ABB RobotStudio station: contour-following.rspag

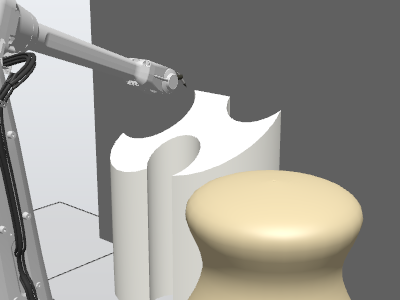
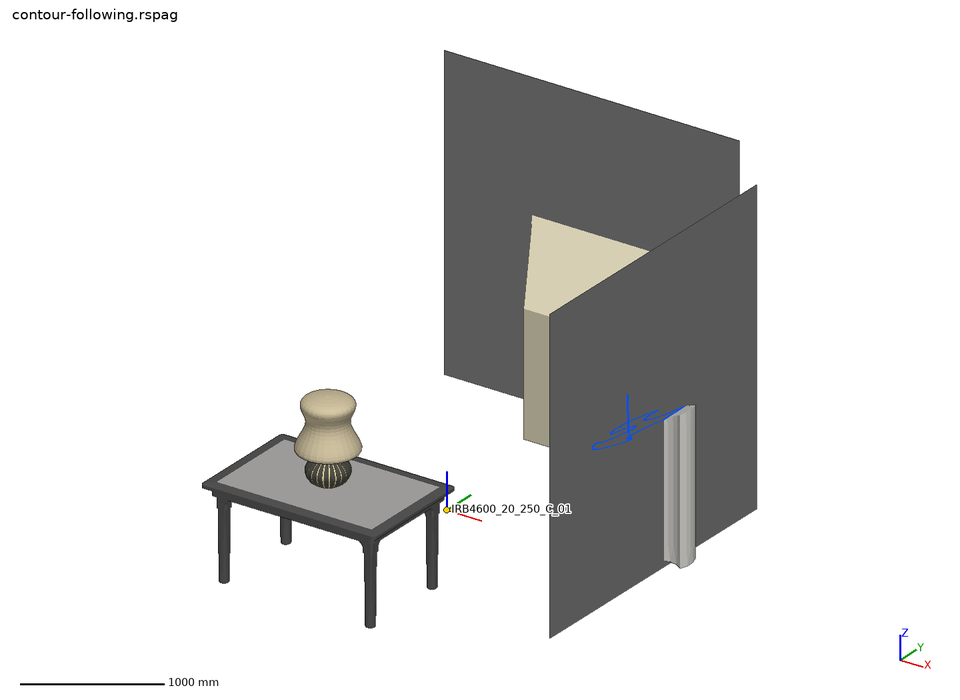
[picture v1: parts stored in the station drawn from their meshes, with robot base, taught points and paths (robot models come from the ABB library and are not in the file)]
--- station ---
Station PenPineappleApplePen (saved by RobotStudio 24.3.10885.0)
Controller Controller2
  mechanical unit ROB_1: IRB4600_20_250_C_01, 6 joints, base frame (0, 0, 0) mm
Layout (positions relative to the parent item):
  - IRB4600_20_250_C_01 [mechanism, from %ABB.RobotStudio.Models.IRB4600%\IRB4600_20_250_C_G_01.rslib] at (0, 0, 0) mm; joint values [0.1057, -0.1541, 0.5189, 0, -0.306, 0] (rad or m)
  - PenPineappleApplePen [mechanism, from Documents\PenPineappleApplePen.rslib] at (1296.51, 137.49, 1296.47) mm, rotated rx 180 ry 86.63 rz -173.95 deg
  - table2 [part] at (1845.28, -943.75, 534.88) mm, rotated rx 90 ry 0 rz 90 deg, size 984.1 x 770.9 x 1476.2 mm
  - trapez [part] at (500, 1748.7, 450) mm, rotated rx 90 ry 0 rz 90 deg, size 606.2 x 1387.4 x 1000 mm
  - krzywik [part] at (2000, 715.02, 706.25) mm, rotated rx 90 ry 0 rz 90 deg, size 823.5 x 1193.4 x 764.8 mm
  - lampa2 [part] at (112.5, -1435.82, 770.92) mm, rotated rx 90 ry 0 rz 90 deg, size 471.7 x 688.5 x 472.4 mm
  - Part_1 [part] at (1745, -1250, 0) mm, size 5 x 2500 x 2500 mm
  - Part_2 [part] at (-1250, 1750, 0) mm, size 2500 x 5 x 2500 mm
  - Frame_2 [frame] at (56.86, 0, 134.14) mm, rotated rx 0 ry 44.94 rz 0 deg
Attachment: PenPineappleApplePen is attached to IRB4600_20_250_C_01 / Link6
Attachment: trapez is attached to trapez
Attachment: krzywik is attached to krzywik
Attachment: lampa is attached to lampa2
Attachment: trapez is attached to Part_2
Attachment: lampa2 is attached to table2
Attachment: krzywik is attached to Part_1
Targets, tools, work objects and paths stored in the station and not in the controller backup, written as RAPID:
! task T_ROB1
MODULE CalibData
  TASK PERS wobjdata trapez:=[FALSE,TRUE,"",[[0,0,50],[1,0,0,0]],[[0,0,0],[1,0,0,0]]];
  TASK PERS wobjdata lampa:=[FALSE,TRUE,"",[[119.9,0,40.518],[1,0,0,0]],[[0,0,0],[1,0,0,0]]];
ENDMODULE

! task T_ROB1
MODULE Module1
  CONST robtarget Target_10:=[[-500,1748.705,1387.429],[0.270478686,-0.652549655,0.65678764,0.263913289],[1,2,1,0],[9E+09,9E+09,9E+09,9E+09,9E+09,9E+09]];
  CONST robtarget Target_20:=[[-150,1142.487,1006.377],[0.270478686,-0.652549655,0.65678764,0.263913289],[1,2,1,0],[9E+09,9E+09,9E+09,9E+09,9E+09,9E+09]];
  CONST robtarget Target_30:=[[150,1142.487,1006.377],[0.270478686,-0.652549655,0.65678764,0.263913289],[0,1,2,0],[9E+09,9E+09,9E+09,9E+09,9E+09,9E+09]];
  CONST robtarget Target_40:=[[500,1748.705,1387.429],[0.270478686,-0.652549655,0.65678764,0.263913289],[0,1,2,0],[9E+09,9E+09,9E+09,9E+09,9E+09,9E+09]];
  CONST robtarget above_trapez:=[[2.354624835,1375.15869908,1439.170310285],[0.270478686,-0.652549655,0.65678764,0.263913289],[1,2,1,0],[9E+09,9E+09,9E+09,9E+09,9E+09,9E+09]];
  CONST robtarget Target_300:=[[1764.521875862,134.170519561,1094.86146005],[0.355319487,-0.049345838,0.933252419,0.018787562],[0,-1,0,1],[9E+09,9E+09,9E+09,9E+09,9E+09,9E+09]];
  CONST robtarget Target_310:=[[1784.700794279,135.94993306,1106.51176403],[0.355319487,-0.049345838,0.933252419,0.018787562],[0,-1,0,1],[9E+09,9E+09,9E+09,9E+09,9E+09,9E+09]];
  CONST robtarget Target_320:=[[1804.953567722,135.525399506,1118.20470823],[0.355319487,-0.049345838,0.933252419,0.018787562],[0,-1,0,1],[9E+09,9E+09,9E+09,9E+09,9E+09,9E+09]];
  CONST robtarget Target_330:=[[1825.040194425,132.901949757,1129.801727564],[0.355319487,-0.049345838,0.933252419,0.018787562],[0,-1,0,1],[9E+09,9E+09,9E+09,9E+09,9E+09,9E+09]];
  CONST robtarget Target_340:=[[1844.722641512,128.110672521,1141.165393688],[0.355319487,-0.049345838,0.933252419,0.018787562],[0,-1,0,1],[9E+09,9E+09,9E+09,9E+09,9E+09,9E+09]];
  CONST robtarget Target_350:=[[1863.767665765,121.208345948,1152.161043566],[0.355319487,-0.049345838,0.933252419,0.018787562],[0,-1,0,1],[9E+09,9E+09,9E+09,9E+09,9E+09,9E+09]];
  CONST robtarget Target_360:=[[1881.949577625,112.276764789,1162.658375273],[0.355319487,-0.049345838,0.933252419,0.018787562],[0,-1,0,1],[9E+09,9E+09,9E+09,9E+09,9E+09,9E+09]];
  CONST robtarget Target_370:=[[1899.052915691,101.421771104,1172.53299211],[0.355319487,-0.049345838,0.933252419,0.018787562],[0,-1,0,1],[9E+09,9E+09,9E+09,9E+09,9E+09,9E+09]];
  CONST robtarget Target_380:=[[1914.875,88.772,1181.667876745],[0.355319487,-0.049345838,0.933252419,0.018787562],[0,-1,0,1],[9E+09,9E+09,9E+09,9E+09,9E+09,9E+09]];
  CONST robtarget Target_390:=[[1924.367037707,112.000280725,1187.14810727],[0.355319487,-0.049345838,0.933252419,0.018787562],[0,-1,0,1],[9E+09,9E+09,9E+09,9E+09,9E+09,9E+09]];
  CONST robtarget Target_400:=[[1930.986602832,136.204271363,1190.969914977],[0.355319487,-0.049345838,0.933252419,0.018787562],[0,-1,0,1],[9E+09,9E+09,9E+09,9E+09,9E+09,9E+09]];
  CONST robtarget Target_410:=[[1934.636942574,161.030201859,1193.07743961],[0.355319487,-0.049345838,0.933252419,0.018787562],[0,-1,0,1],[9E+09,9E+09,9E+09,9E+09,9E+09,9E+09]];
  CONST robtarget Target_420:=[[1935.264702885,186.11521177,1193.439877194],[0.355319487,-0.049345838,0.933252419,0.018787562],[0,-1,0,1],[9E+09,9E+09,9E+09,9E+09,9E+09,9E+09]];
  CONST robtarget Target_430:=[[1932.860708302,211.092653899,1192.051930274],[0.355319487,-0.049345838,0.933252419,0.018787562],[0,0,-1,1],[9E+09,9E+09,9E+09,9E+09,9E+09,9E+09]];
  CONST robtarget Target_440:=[[1927.460096059,235.597453279,1188.933885342],[0.355319487,-0.049345838,0.933252419,0.018787562],[0,0,-1,1],[9E+09,9E+09,9E+09,9E+09,9E+09,9E+09]];
  CONST robtarget Target_450:=[[1919.141802515,259.271443179,1184.131316326],[0.355319487,-0.049345838,0.933252419,0.018787562],[0,0,-1,1],[9E+09,9E+09,9E+09,9E+09,9E+09,9E+09]];
  CONST robtarget Target_460:=[[1908.027409406,281.768600134,1177.714418472],[0.355319487,-0.049345838,0.933252419,0.018787562],[0,0,-1,1],[9E+09,9E+09,9E+09,9E+09,9E+09,9E+09]];
  CONST robtarget Target_470:=[[1894.279366779,302.76010149,1169.77698236],[0.355319487,-0.049345838,0.933252419,0.018787562],[0,0,-1,1],[9E+09,9E+09,9E+09,9E+09,9E+09,9E+09]];
  CONST robtarget Target_480:=[[1878.098618597,321.939131536,1160.435023042],[0.355319487,-0.049345838,0.933252419,0.018787562],[0,0,-1,1],[9E+09,9E+09,9E+09,9E+09,9E+09,9E+09]];
  CONST robtarget Target_490:=[[1859.721665702,339.025365983,1149.825084341],[0.355319487,-0.049345838,0.933252419,0.018787562],[0,0,-1,1],[9E+09,9E+09,9E+09,9E+09,9E+09,9E+09]];
  CONST robtarget Target_500:=[[1839.417109075,353.76906923,1138.102243107],[0.355319487,-0.049345838,0.933252419,0.018787562],[0,0,-1,1],[9E+09,9E+09,9E+09,9E+09,9E+09,9E+09]];
  CONST robtarget Target_510:=[[1817.481723914,365.954744554,1125.43784258],[0.355319487,-0.049345838,0.933252419,0.018787562],[0,0,-1,1],[9E+09,9E+09,9E+09,9E+09,9E+09,9E+09]];
  CONST robtarget Target_520:=[[1794.236121912,375.404283845,1112.016988006],[0.355319487,-0.049345838,0.933252419,0.018787562],[0,0,-1,1],[9E+09,9E+09,9E+09,9E+09,9E+09,9E+09]];
  CONST robtarget Target_530:=[[1770.020065136,381.979570869,1098.035841107],[0.355319487,-0.049345838,0.933252419,0.018787562],[0,0,-1,1],[9E+09,9E+09,9E+09,9E+09,9E+09,9E+09]];
  CONST robtarget Target_1470:=[[-356.227701034,-1435.823,1008.367912023],[0,0.5726162,0,0.819823571],[-2,0,0,0],[9E+09,9E+09,9E+09,9E+09,9E+09,9E+09]];
  CONST robtarget Target_1480:=[[-356.632819707,-1435.823,1024.985425278],[0,0.7722597,0,0.635306978],[-2,0,0,0],[9E+09,9E+09,9E+09,9E+09,9E+09,9E+09]];
  CONST robtarget Target_1490:=[[-349.496807665,-1435.823,1046.554535488],[0,0.834440548,0,0.55109797],[-2,0,0,0],[9E+09,9E+09,9E+09,9E+09,9E+09,9E+09]];
  CONST robtarget Target_1500:=[[-337.487544389,-1435.823,1071.313546721],[0,0.856155357,0,0.516718497],[-2,0,0,0],[9E+09,9E+09,9E+09,9E+09,9E+09,9E+09]];
  CONST robtarget Target_1510:=[[-308.314339892,-1435.823,1124.876064439],[0,0.855906278,0,0.517130974],[-2,0,0,0],[9E+09,9E+09,9E+09,9E+09,9E+09,9E+09]];
  CONST robtarget Target_1520:=[[-285.046138139,-1435.823,1178.110750529],[0,0.805538472,0,0.592543476],[-2,0,0,0],[9E+09,9E+09,9E+09,9E+09,9E+09,9E+09]];
  CONST robtarget Target_1530:=[[-279.294170946,-1435.823,1203.768042628],[0,0.750595327,0,0.660762177],[-2,0,0,0],[9E+09,9E+09,9E+09,9E+09,9E+09,9E+09]];
  CONST robtarget Target_1540:=[[-278.820319707,-1435.823,1229.036477464],[0,0.672760595,0,0.739860245],[-2,0,0,0],[9E+09,9E+09,9E+09,9E+09,9E+09,9E+09]];
  CONST robtarget Target_1550:=[[-284.181369532,-1435.823,1254.504702787],[0,0.590226841,0,0.807237435],[-2,0,0,0],[9E+09,9E+09,9E+09,9E+09,9E+09,9E+09]];
  CONST robtarget Target_1560:=[[-316.030461305,-1435.823,1334.787935859],[0,0.640987484,0,0.767551331],[-2,0,0,0],[9E+09,9E+09,9E+09,9E+09,9E+09,9E+09]];
  CONST robtarget Target_1570:=[[-313.831298622,-1435.823,1361.259758709],[0,0.834769365,0,0.550599771],[-2,0,0,0],[9E+09,9E+09,9E+09,9E+09,9E+09,9E+09]];
  CONST robtarget Target_1580:=[[-305.449627822,-1435.823,1373.780481427],[0,0.918497838,0,0.395425999],[-2,0,0,0],[9E+09,9E+09,9E+09,9E+09,9E+09,9E+09]];
  CONST robtarget Target_1590:=[[-290.274693372,-1435.823,1385.522452993],[0,0.964723418,0,0.263265506],[-2,-1,0,0],[9E+09,9E+09,9E+09,9E+09,9E+09,9E+09]];
  CONST robtarget Target_1600:=[[-266.667771673,-1435.823,1396.219409162],[0,0.985506762,0,0.169636146],[-2,-1,0,0],[9E+09,9E+09,9E+09,9E+09,9E+09,9E+09]];
  CONST robtarget Target_1610:=[[-232.842282653,-1435.823,1405.5732495],[0,0.994311989,0,0.106506661],[-2,-1,1,0],[9E+09,9E+09,9E+09,9E+09,9E+09,9E+09]];
  CONST robtarget Target_1620:=[[-186.863789768,-1435.823,1413.254037383],[0,0.997988983,0,0.063387614],[-1,-1,1,0],[9E+09,9E+09,9E+09,9E+09,9E+09,9E+09]];
  CONST robtarget Target_1630:=[[-126.65,-1435.823,1418.9],[0,0.999455226,0,0.033003814],[-1,-1,1,0],[9E+09,9E+09,9E+09,9E+09,9E+09,9E+09]];
  CONST robtarget Target_1640:=[[-129.948583459,-1435.823,1468.791074825],[0,0.999455226,0,0.033003814],[-1,-1,1,0],[9E+09,9E+09,9E+09,9E+09,9E+09,9E+09]];
  CONST robtarget above_lamp:=[[-394.039408817,-1297.199647583,1588.358827541],[0.508942412,0.79207847,0.336817323,-0.011975388],[-2,-1,1,0],[9E+09,9E+09,9E+09,9E+09,9E+09,9E+09]];
  CONST robtarget back_trace:=[[-404.928368365,-1011.661568461,885.919207147],[0.385577292,0.834726208,0.074942636,0.385935112],[-2,0,0,0],[9E+09,9E+09,9E+09,9E+09,9E+09,9E+09]];
  CONST robtarget Target_1650:=[[1079.225,237.179079749,785.646448491],[0.101814374,0.888048773,0.379976418,0.237951952],[0,0,0,0],[9E+09,9E+09,9E+09,9E+09,9E+09,9E+09]];
  CONST robtarget Target_1660:=[[1104.225,237.179079749,742.345178302],[0.101814374,0.888048773,0.379976418,0.237951952],[0,-1,1,0],[9E+09,9E+09,9E+09,9E+09,9E+09,9E+09]];
  CONST robtarget Target_1670:=[[1135.277965809,264.790385883,760.273616471],[0.065302717,0.934674621,0.243713057,0.25044531],[0,-1,1,0],[9E+09,9E+09,9E+09,9E+09,9E+09,9E+09]];
  CONST robtarget Target_1680:=[[1173.212092282,281.751310408,782.174894602],[0.030064157,0.95938712,0.112200961,0.257067004],[0,-1,2,0],[9E+09,9E+09,9E+09,9E+09,9E+09,9E+09]];
  CONST robtarget Target_1690:=[[1214.495098447,286.482516812,806.009649324],[0.004378616,-0.965787589,0.016341217,-0.258782004],[0,0,2,0],[9E+09,9E+09,9E+09,9E+09,9E+09,9E+09]];
  CONST robtarget Target_1700:=[[1255.282868444,278.543453224,829.558479312],[0.038945016,-0.954928058,0.14534478,-0.255872202],[0,0,2,0],[9E+09,9E+09,9E+09,9E+09,9E+09,9E+09]];
  CONST robtarget Target_1710:=[[1291.777400916,258.673374924,850.628607458],[0.074493857,-0.925051588,0.278014857,-0.247866826],[0,0,2,0],[9E+09,9E+09,9E+09,9E+09,9E+09,9E+09]];
  CONST robtarget Target_1720:=[[1320.580464386,228.722507712,867.258063906],[0.111291008,-0.872067838,0.415343698,-0.233669873],[0,0,2,0],[9E+09,9E+09,9E+09,9E+09,9E+09,9E+09]];
  CONST robtarget Target_1730:=[[1339.010027592,191.479761948,877.898377184],[0.148334096,-0.79154936,0.553590384,-0.212095012],[0,0,2,0],[9E+09,9E+09,9E+09,9E+09,9E+09,9E+09]];
  CONST robtarget Target_1740:=[[1345.35,150.413039874,881.558761961],[0.183012702,-0.683012702,0.683012702,-0.183012702],[0,0,2,0],[9E+09,9E+09,9E+09,9E+09,9E+09,9E+09]];
  CONST robtarget Target_1750:=[[1339.010027592,109.346317801,877.898377184],[0.212095012,-0.553590384,0.79154936,-0.148334096],[0,0,2,0],[9E+09,9E+09,9E+09,9E+09,9E+09,9E+09]];
  CONST robtarget Target_1760:=[[1320.580464386,72.103572037,867.258063906],[0.233669873,-0.415343698,0.872067838,-0.111291008],[-1,1,2,0],[9E+09,9E+09,9E+09,9E+09,9E+09,9E+09]];
  CONST robtarget Target_1770:=[[1291.777400916,42.152704825,850.628607458],[0.247866826,-0.278014857,0.925051588,-0.074493857],[-1,1,2,0],[9E+09,9E+09,9E+09,9E+09,9E+09,9E+09]];
  CONST robtarget Target_1780:=[[1255.282868444,22.282626525,829.558479312],[0.255872202,-0.14534478,0.954928058,-0.038945016],[-1,1,2,0],[9E+09,9E+09,9E+09,9E+09,9E+09,9E+09]];
  CONST robtarget Target_1790:=[[1214.495098447,14.343562937,806.009649324],[0.258782004,-0.016341217,0.965787589,-0.004378616],[0,1,2,0],[9E+09,9E+09,9E+09,9E+09,9E+09,9E+09]];
  CONST robtarget Target_1800:=[[1173.212092282,19.074769341,782.174894602],[0.257067004,0.112200961,0.95938712,0.030064157],[0,2,1,0],[9E+09,9E+09,9E+09,9E+09,9E+09,9E+09]];
  CONST robtarget Target_1810:=[[1135.277965809,36.035693866,760.273616471],[0.25044531,0.243713057,0.934674621,0.065302717],[0,2,1,0],[9E+09,9E+09,9E+09,9E+09,9E+09,9E+09]];
  CONST robtarget Target_1820:=[[1104.225,63.647,742.345178302],[0.237951952,0.379976418,0.888048773,0.101814374],[0,2,1,0],[9E+09,9E+09,9E+09,9E+09,9E+09,9E+09]];
  CONST robtarget Target_1830:=[[1115.168705531,24.942095166,748.663529636],[0.145865677,-0.797913008,0.544378117,-0.213800146],[-1,0,2,0],[9E+09,9E+09,9E+09,9E+09,9E+09,9E+09]];
  CONST robtarget Target_1840:=[[1130.03531583,-12.431936557,757.246771094],[0.133473684,-0.827573947,0.498130569,-0.221747771],[-1,0,2,0],[9E+09,9E+09,9E+09,9E+09,9E+09,9E+09]];
  CONST robtarget Target_1850:=[[1148.667140429,-48.078667979,768.003860042],[0.120964856,-0.853936951,0.45144699,-0.228811716],[-1,0,2,0],[9E+09,9E+09,9E+09,9E+09,9E+09,9E+09]];
  CONST robtarget Target_1860:=[[1170.86655115,-81.619993425,780.820695798],[0.108438136,-0.877059483,0.404696634,-0.23500738],[-1,0,2,0],[9E+09,9E+09,9E+09,9E+09,9E+09,9E+09]];
  CONST robtarget Target_1870:=[[1196.398078347,-112.700139306,795.561329898],[0.095969627,-0.897068332,0.358163523,-0.240368735],[-1,0,2,0],[9E+09,9E+09,9E+09,9E+09,9E+09,9E+09]];
  CONST robtarget Target_1880:=[[1224.990908541,-140.989437821,812.069408107],[0.083611988,-0.914134086,0.312044187,-0.24494149],[-1,0,2,0],[9E+09,9E+09,9E+09,9E+09,9E+09,9E+09]];
  CONST robtarget Target_1890:=[[1256.341756944,-166.187823749,830.169828872],[0.071395991,-0.928447766,0.266453464,-0.248776829],[-1,0,2,0],[9E+09,9E+09,9E+09,9E+09,9E+09,9E+09]];
  CONST robtarget Target_1900:=[[1290.118084407,-188.028017249,849.670600625],[0.059333361,-0.940201676,0.221435117,-0.25192628],[-1,0,2,0],[9E+09,9E+09,9E+09,9E+09,9E+09,9E+09]];
  CONST robtarget Target_1910:=[[1325.96162467,-206.2783589,870.364878245],[0.047420169,-0.949575029,0.17697448,-0.254437862],[-1,0,2,0],[9E+09,9E+09,9E+09,9E+09,9E+09,9E+09]];
  CONST robtarget Target_1920:=[[1363.492184502,-220.745266921,892.033157066],[0.035640235,-0.956723957,0.133011169,-0.256353412],[-1,0,1,0],[9E+09,9E+09,9E+09,9E+09,9E+09,9E+09]];
  CONST robtarget Target_1930:=[[1402.311676416,-231.275290496,914.445601173],[0.023968254,-0.96177506,0.089450741,-0.257706851],[-1,0,1,0],[9E+09,9E+09,9E+09,9E+09,9E+09,9E+09]];
  CONST robtarget Target_1940:=[[1442.008341196,-237.756737429,937.36448127],[0.012372518,-0.964821529,0.046174865,-0.25852315],[-1,0,1,0],[9E+09,9E+09,9E+09,9E+09,9E+09,9E+09]];
  CONST robtarget Target_1950:=[[1482.161115432,-240.120858867,960.546696283],[0.000817262,-0.965921011,0.003050063,-0.258817755],[-1,-1,1,0],[9E+09,9E+09,9E+09,9E+09,9E+09,9E+09]];
  CONST robtarget Target_1960:=[[1522.34409775,-238.342578523,983.746351942],[0.010735293,0.965094568,0.04006466,0.25859631],[-1,-1,1,0],[9E+09,9E+09,9E+09,9E+09,9E+09,9E+09]];
  CONST robtarget Target_1970:=[[1562.131066361,-232.440758656,1006.717368979],[0.022323059,0.962326355,0.08331079,0.25785457],[-1,-1,1,0],[9E+09,9E+09,9E+09,9E+09,9E+09,9E+09]];
  CONST robtarget Target_1980:=[[1601.1,-222.478,1029.216093306],[0.033982204,0.957563862,0.126823313,0.256578463],[-1,-1,1,0],[9E+09,9E+09,9E+09,9E+09,9E+09,9E+09]];
  CONST robtarget Target_1990:=[[1565.485723439,-203.289964368,1008.654181146],[0.249518515,0.256612319,0.931215775,0.068759064],[-1,-2,1,0],[9E+09,9E+09,9E+09,9E+09,9E+09,9E+09]];
  CONST robtarget Target_2000:=[[1534.859704885,-176.858838892,990.97224109],[0.240877448,0.353371284,0.898966872,0.09468555],[-1,-2,1,0],[9E+09,9E+09,9E+09,9E+09,9E+09,9E+09]];
  CONST robtarget Target_2010:=[[1510.669355527,-144.433780614,977.005936376],[0.228741176,0.45194461,0.853673691,0.121098193],[-1,-1,1,0],[9E+09,9E+09,9E+09,9E+09,9E+09,9E+09]];
  CONST robtarget Target_2020:=[[1494.057931457,-107.547224842,967.415326218],[0.212747139,0.550094071,0.793983133,0.147397262],[-1,-1,1,0],[9E+09,9E+09,9E+09,9E+09,9E+09,9E+09]];
  CONST robtarget Target_2030:=[[1485.810502435,-67.942460975,962.653670852],[0.192899661,0.644003393,0.719911336,0.172560189],[0,-1,1,0],[9E+09,9E+09,9E+09,9E+09,9E+09,9E+09]];
  CONST robtarget Target_2040:=[[1486.31684884,-27.491243198,962.946010085],[0.169765377,0.729107632,0.633573014,0.195363801],[0,-1,1,0],[9E+09,9E+09,9E+09,9E+09,9E+09,9E+09]];
  CONST robtarget Target_2050:=[[1495.553040316,11.89467019,968.27852772],[0.144410213,0.80159194,0.538946253,0.214785913],[0,-1,1,0],[9E+09,9E+09,9E+09,9E+09,9E+09,9E+09]];
  CONST robtarget Target_2060:=[[1513.082566748,48.353868061,978.399204525],[0.118053068,0.859594046,0.440580048,0.23032753],[0,-1,1,0],[9E+09,9E+09,9E+09,9E+09,9E+09,9E+09]];
  CONST robtarget Target_2070:=[[1538.076968094,80.163258307,992.82972887],[0.091674424,0.903303545,0.342133609,0.242039456],[0,-1,1,0],[9E+09,9E+09,9E+09,9E+09,9E+09,9E+09]];
  CONST robtarget Target_2080:=[[1569.354988092,105.819502603,1010.888102135],[0.065822324,0.934166832,0.245652257,0.250309248],[0,-1,1,0],[9E+09,9E+09,9E+09,9E+09,9E+09,9E+09]];
  CONST robtarget Target_2090:=[[1605.43840142,124.110065441,1031.720870534],[0.040637159,0.953945472,0.151659942,0.255608919],[0,-1,1,0],[9E+09,9E+09,9E+09,9E+09,9E+09,9E+09]];
  CONST robtarget Target_2100:=[[1644.621875862,134.170519561,1054.34346005],[0.015977034,0.964083664,0.059627104,0.258325439],[0,-1,1,0],[9E+09,9E+09,9E+09,9E+09,9E+09,9E+09]];
  CONST robtarget Target_2110:=[[1685.053567722,135.525399506,1077.68670823],[0.008454424,-0.965410354,0.031552341,-0.258680925],[0,0,2,0],[9E+09,9E+09,9E+09,9E+09,9E+09,9E+09]];
  CONST robtarget Target_2120:=[[1724.822641512,128.110672521,1100.647393688],[0.033008401,-0.958038186,0.123189029,-0.256705558],[0,0,2,0],[9E+09,9E+09,9E+09,9E+09,9E+09,9E+09]];
  CONST robtarget Target_2130:=[[1762.049577625,112.276764789,1122.140375273],[0.058007536,-0.941353307,0.216487073,-0.252234858],[0,0,2,0],[9E+09,9E+09,9E+09,9E+09,9E+09,9E+09]];
  CONST robtarget Target_2140:=[[1794.975,88.772,1141.149876745],[0.083653614,-0.914081041,0.312199539,-0.244927277],[0,0,2,0],[9E+09,9E+09,9E+09,9E+09,9E+09,9E+09]];
  CONST robtarget Target_2150:=[[1811.086602832,136.204271363,1150.451914977],[0.160061595,0.759062655,0.597358006,0.203390226],[0,-1,1,0],[9E+09,9E+09,9E+09,9E+09,9E+09,9E+09]];
  CONST robtarget Target_2160:=[[1815.364702885,186.11521177,1152.921877194],[0.186720933,0.668887119,0.69685201,0.179227763],[0,-1,1,0],[9E+09,9E+09,9E+09,9E+09,9E+09,9E+09]];
  CONST robtarget Target_2170:=[[1807.560096059,235.597453279,1148.415885342],[0.209655409,0.566385989,0.782444639,0.151762668],[0,-1,1,0],[9E+09,9E+09,9E+09,9E+09,9E+09,9E+09]];
  CONST robtarget Target_2180:=[[1788.127409406,281.768600134,1137.196418472],[0.227916914,0.457707976,0.850597502,0.122642482],[0,-1,1,0],[9E+09,9E+09,9E+09,9E+09,9E+09,9E+09]];
  CONST robtarget Target_2190:=[[1758.198618597,321.939131536,1119.917023042],[0.241413165,0.348242177,0.900966197,0.09331121],[0,-1,1,0],[9E+09,9E+09,9E+09,9E+09,9E+09,9E+09]];
  CONST robtarget Target_2200:=[[1719.517109075,353.76906923,1097.584243107],[0.250629262,0.241064801,0.935361141,0.064593119],[0,-2,1,0],[9E+09,9E+09,9E+09,9E+09,9E+09,9E+09]];
  CONST robtarget Target_2210:=[[1674.336121912,375.404283845,1071.498988006],[0.25620536,0.136926686,0.95617142,0.036689395],[0,-2,1,0],[9E+09,9E+09,9E+09,9E+09,9E+09,9E+09]];
  CONST robtarget Target_2220:=[[1625.2875,385.5845,1043.180752942],[0.258648972,0.035011232,0.965291104,0.009381231],[0,-2,1,0],[9E+09,9E+09,9E+09,9E+09,9E+09,9E+09]];
  CONST robtarget Target_2230:=[[1601.044864766,356.220958453,1029.184260964],[0.242378357,-0.338775461,0.904568344,-0.090774611],[0,-3,2,0],[9E+09,9E+09,9E+09,9E+09,9E+09,9E+09]];
  CONST robtarget Target_2240:=[[1571.827205325,331.802700693,1012.31543742],[0.249492039,-0.256970612,0.931116967,-0.068855068],[0,-3,2,0],[9E+09,9E+09,9E+09,9E+09,9E+09,9E+09]];
  CONST robtarget Target_2250:=[[1538.626094744,313.158420299,993.146767289],[0.25443798,-0.176972116,0.949575469,-0.047419536],[0,-3,2,0],[9E+09,9E+09,9E+09,9E+09,9E+09,9E+09]];
  CONST robtarget Target_2260:=[[1502.568294293,300.920856738,972.328786492],[0.257468504,-0.098547878,0.960885538,-0.026405824],[0,-2,1,0],[9E+09,9E+09,9E+09,9E+09,9E+09,9E+09]];
  CONST robtarget Target_2270:=[[1464.877514033,295.505321802,950.568004363],[0.258757227,-0.021110286,0.965695116,-0.005656484],[0,-2,1,0],[9E+09,9E+09,9E+09,9E+09,9E+09,9E+09]];
  CONST robtarget Target_2280:=[[1426.832883206,297.095604975,928.602926514],[0.25838206,0.056106136,0.964294977,0.015033594],[0,-2,1,0],[9E+09,9E+09,9E+09,9E+09,9E+09,9E+09]];
  CONST robtarget Target_2290:=[[1389.725539846,305.63773609,907.178991836],[0.256320082,0.133902818,0.95659957,0.035879152],[0,-2,1,0],[9E+09,9E+09,9E+09,9E+09,9E+09,9E+09]];
  CONST robtarget Target_2300:=[[1354.814812829,320.841816939,887.023274195],[0.25244889,0.212983924,0.942152084,0.057068871],[0,-2,1,0],[9E+09,9E+09,9E+09,9E+09,9E+09,9E+09]];
  CONST robtarget Target_2310:=[[1323.285483462,342.191859676,868.819807398],[0.246556037,0.293800792,0.920159658,0.078723685],[0,-2,1,0],[9E+09,9E+09,9E+09,9E+09,9E+09,9E+09]];
  CONST robtarget Target_2320:=[[1296.20757701,368.96329814,853.186370819],[0.238364885,0.376354326,0.889589862,0.100843838],[0,-2,1,0],[9E+09,9E+09,9E+09,9E+09,9E+09,9E+09]];
  CONST robtarget Target_2330:=[[1274.500048766,400.247577783,840.653523543],[0.227589702,0.459970159,0.849376333,0.123248633],[0,-1,1,0],[9E+09,9E+09,9E+09,9E+09,9E+09,9E+09]];
  CONST robtarget Target_2340:=[[1258.899597041,434.982989703,831.646598541],[0.214028605,0.543126297,0.798765627,0.145530253],[0,-1,1,0],[9E+09,9E+09,9E+09,9E+09,9E+09,9E+09]];
  CONST robtarget Target_2350:=[[1249.935661499,471.990702344,826.471267943],[0.197680828,0.623482494,0.737754893,0.167061631],[0,-1,1,0],[9E+09,9E+09,9E+09,9E+09,9E+09,9E+09]];
  CONST robtarget Target_2360:=[[1247.912455319,510.014768039,825.30316931],[0.178837583,0.698246829,0.667430946,0.187094674],[0,-1,1,0],[9E+09,9E+09,9E+09,9E+09,9E+09,9E+09]];
  CONST robtarget Target_2370:=[[1252.898640973,547.764746686,828.181944939],[0.158077387,0.764832237,0.589952838,0.20493618],[0,-1,1,0],[9E+09,9E+09,9E+09,9E+09,9E+09,9E+09]];
  CONST robtarget Target_2380:=[[1264.725,583.9595,835.009896507],[0.136140408,0.821501337,0.508082921,0.22012062],[0,-1,1,0],[9E+09,9E+09,9E+09,9E+09,9E+09,9E+09]];
  CONST robtarget Target_2390:=[[1234.428871964,582.733933377,817.51841883],[0.258505543,-0.047528015,0.964755819,-0.012735093],[0,-2,1,0],[9E+09,9E+09,9E+09,9E+09,9E+09,9E+09]];
  CONST robtarget Target_2400:=[[1204.634785103,577.106342805,800.316794761],[0.257164531,-0.109043723,0.959751097,-0.029218177],[0,-2,1,0],[9E+09,9E+09,9E+09,9E+09,9E+09,9E+09]];
  CONST robtarget Target_2410:=[[1175.978894374,567.196887017,783.772308534],[0.254719351,-0.171241772,0.950625561,-0.045884095],[0,-2,1,0],[9E+09,9E+09,9E+09,9E+09,9E+09,9E+09]];
  CONST robtarget Target_2420:=[[1149.073052289,553.217149921,768.238213364],[0.251081735,-0.234414993,0.937049792,-0.062811308],[0,-2,1,0],[9E+09,9E+09,9E+09,9E+09,9E+09,9E+09]];
  CONST robtarget Target_2430:=[[1124.491744818,535.46562293,754.046188878],[0.24613106,-0.298722627,0.918573619,-0.080042487],[0,-3,1,0],[9E+09,9E+09,9E+09,9E+09,9E+09,9E+09]];
  CONST robtarget Target_2440:=[[1102.759825117,514.321331652,741.499259189],[0.239725003,-0.364123117,0.894665892,-0.097566495],[0,-3,1,0],[9E+09,9E+09,9E+09,9E+09,9E+09,9E+09]];
  CONST robtarget Target_2450:=[[1084.34130702,490.235743044,730.865322808],[0.231718435,-0.430301818,0.864784972,-0.115299025],[0,-3,2,0],[9E+09,9E+09,9E+09,9E+09,9E+09,9E+09]];
  CONST robtarget Target_2460:=[[1069.629457541,463.723125813,722.371432551],[0.221992238,-0.496611654,0.828486311,-0.133066692],[0,-3,2,0],[9E+09,9E+09,9E+09,9E+09,9E+09,9E+09]];
  CONST robtarget Target_2470:=[[1058.93839995,435.349569901,716.198947572],[0.210490143,-0.562057232,0.785559909,-0.150602781],[0,-3,2,0],[9E+09,9E+09,9E+09,9E+09,9E+09,9E+09]];
  CONST robtarget Target_2480:=[[1052.496406698,405.720899487,712.479661035],[0.19725541,-0.625356329,0.736167212,-0.167563723],[0,-4,2,0],[9E+09,9E+09,9E+09,9E+09,9E+09,9E+09]];
  CONST robtarget Target_2490:=[[1050.441025414,375.469737604,711.292986097],[0.182453249,-0.685094245,0.680924795,-0.18357045],[0,-4,2,0],[9E+09,9E+09,9E+09,9E+09,9E+09,9E+09]];
  CONST robtarget Target_2500:=[[1052.816142018,345.241998545,712.664260308],[0.166364969,-0.739944323,0.620882518,-0.198267484],[0,-4,2,0],[9E+09,9E+09,9E+09,9E+09,9E+09,9E+09]];
  CONST robtarget Target_2510:=[[1059.571043691,315.683096486,716.564204607],[0.149349844,-0.788884587,0.557381207,-0.211380988],[0,-4,2,0],[9E+09,9E+09,9E+09,9E+09,9E+09,9E+09]];
  CONST robtarget Target_2520:=[[1070.561501673,287.424164785,722.909548481],[0.131786232,-0.831332116,0.491832913,-0.222754769],[0,-4,2,0],[9E+09,9E+09,9E+09,9E+09,9E+09,9E+09]];
  CONST robtarget Target_2530:=[[1085.552850798,261.068580198,731.564807934],[0.114013243,-0.867156107,0.425503217,-0.232353779],[0,-4,2,0],[9E+09,9E+09,9E+09,9E+09,9E+09,9E+09]];
  CONST robtarget Target_2540:=[[1104.225,237.179079749,742.345178302],[0.096291106,-0.896588379,0.3593633,-0.240240132],[0,-4,2,0],[9E+09,9E+09,9E+09,9E+09,9E+09,9E+09]];
  CONST robtarget Target_2550:=[[1079.225,237.179079749,785.646448491],[0.096291106,-0.896588379,0.3593633,-0.240240132],[0,-4,2,0],[9E+09,9E+09,9E+09,9E+09,9E+09,9E+09]];
  LOCAL PROC Path_10()
    MoveL above_trapez,v1000,fine,PenPineappleApplePen\WObj:=trapez;
    MoveL Target_10,v1000,fine,PenPineappleApplePen\WObj:=trapez;
    MoveL Target_20,v300,fine,PenPineappleApplePen\WObj:=trapez;
    MoveL Target_30,v300,fine,PenPineappleApplePen\WObj:=trapez;
    MoveL Target_40,v300,fine,PenPineappleApplePen\WObj:=trapez;
    MoveL Target_10,v300,fine,PenPineappleApplePen\WObj:=trapez;
    MoveL above_trapez,v1000,fine,PenPineappleApplePen\WObj:=trapez;
  ENDPROC
  PROC Path_20()
    MoveL above_krzywik,v1000,z100,PenPineappleApplePen\WObj:=krzywik;
    MoveL Target_50,v1000,z100,PenPineappleApplePen\WObj:=krzywik;
    MoveL Target_60,v300,fine,PenPineappleApplePen\WObj:=krzywik;
    MoveL Target_70,v300,z100,PenPineappleApplePen\WObj:=krzywik;
    MoveL Target_80,v300,z100,PenPineappleApplePen\WObj:=krzywik;
    MoveL Target_90,v300,z100,PenPineappleApplePen\WObj:=krzywik;
    MoveL Target_100,v300,z100,PenPineappleApplePen\WObj:=krzywik;
    MoveL Target_110,v300,z100,PenPineappleApplePen\WObj:=krzywik;
    MoveL Target_120,v300,z100,PenPineappleApplePen\WObj:=krzywik;
    MoveL Target_130,v300,z100,PenPineappleApplePen\WObj:=krzywik;
    MoveL Target_140,v300,z100,PenPineappleApplePen\WObj:=krzywik;
    MoveL Target_150,v300,z100,PenPineappleApplePen\WObj:=krzywik;
    MoveL Target_160,v300,z100,PenPineappleApplePen\WObj:=krzywik;
    MoveL Target_170,v300,z100,PenPineappleApplePen\WObj:=krzywik;
    MoveL Target_180,v300,z100,PenPineappleApplePen\WObj:=krzywik;
    MoveL Target_190,v300,z100,PenPineappleApplePen\WObj:=krzywik;
    MoveL Target_200,v300,z100,PenPineappleApplePen\WObj:=krzywik;
    MoveL Target_210,v300,z100,PenPineappleApplePen\WObj:=krzywik;
    MoveL Target_220,v300,z100,PenPineappleApplePen\WObj:=krzywik;
    MoveL Target_230,v300,z100,PenPineappleApplePen\WObj:=krzywik;
    MoveL Target_240,v300,z100,PenPineappleApplePen\WObj:=krzywik;
    MoveL Target_250,v300,z100,PenPineappleApplePen\WObj:=krzywik;
    MoveL Target_260,v300,z100,PenPineappleApplePen\WObj:=krzywik;
    MoveL Target_270,v300,z100,PenPineappleApplePen\WObj:=krzywik;
    MoveL Target_280,v300,z100,PenPineappleApplePen\WObj:=krzywik;
    MoveL Target_290,v300,z100,PenPineappleApplePen\WObj:=krzywik;
    MoveL Target_540,v300,z100,PenPineappleApplePen\WObj:=krzywik;
    MoveL Target_550,v300,z100,PenPineappleApplePen\WObj:=krzywik;
    MoveL Target_560,v300,z100,PenPineappleApplePen\WObj:=krzywik;
    MoveL Target_570,v300,z100,PenPineappleApplePen\WObj:=krzywik;
    MoveL Target_580,v300,z100,PenPineappleApplePen\WObj:=krzywik;
    MoveL Target_590,v300,z100,PenPineappleApplePen\WObj:=krzywik;
    MoveL Target_600,v300,z100,PenPineappleApplePen\WObj:=krzywik;
    MoveL Target_610,v300,z100,PenPineappleApplePen\WObj:=krzywik;
    MoveL Target_620,v300,z100,PenPineappleApplePen\WObj:=krzywik;
    MoveL Target_630,v300,z100,PenPineappleApplePen\WObj:=krzywik;
    MoveL Target_640,v300,z100,PenPineappleApplePen\WObj:=krzywik;
    MoveL Target_650,v300,z100,PenPineappleApplePen\WObj:=krzywik;
    MoveL Target_660,v300,z100,PenPineappleApplePen\WObj:=krzywik;
    MoveL Target_670,v300,z100,PenPineappleApplePen\WObj:=krzywik;
    MoveL Target_680,v300,z100,PenPineappleApplePen\WObj:=krzywik;
    MoveL Target_690,v300,z100,PenPineappleApplePen\WObj:=krzywik;
    MoveL Target_700,v300,z100,PenPineappleApplePen\WObj:=krzywik;
    MoveL Target_710,v300,z100,PenPineappleApplePen\WObj:=krzywik;
    MoveL Target_720,v300,z100,PenPineappleApplePen\WObj:=krzywik;
    MoveL Target_730,v300,z100,PenPineappleApplePen\WObj:=krzywik;
    MoveL Target_740,v300,z100,PenPineappleApplePen\WObj:=krzywik;
    MoveL Target_750,v300,z100,PenPineappleApplePen\WObj:=krzywik;
    MoveL Target_760,v300,z100,PenPineappleApplePen\WObj:=krzywik;
    MoveL Target_770,v300,z100,PenPineappleApplePen\WObj:=krzywik;
    MoveL Target_780,v300,z100,PenPineappleApplePen\WObj:=krzywik;
    MoveL Target_790,v300,z100,PenPineappleApplePen\WObj:=krzywik;
    MoveL Target_800,v300,z100,PenPineappleApplePen\WObj:=krzywik;
    MoveL Target_810,v300,z100,PenPineappleApplePen\WObj:=krzywik;
    MoveL Target_820,v300,z100,PenPineappleApplePen\WObj:=krzywik;
    MoveL Target_830,v300,z100,PenPineappleApplePen\WObj:=krzywik;
    MoveL Target_840,v300,z100,PenPineappleApplePen\WObj:=krzywik;
    MoveL Target_850,v300,z100,PenPineappleApplePen\WObj:=krzywik;
    MoveL Target_860,v300,z100,PenPineappleApplePen\WObj:=krzywik;
    MoveL Target_870,v300,z100,PenPineappleApplePen\WObj:=krzywik;
    MoveL Target_880,v300,z100,PenPineappleApplePen\WObj:=krzywik;
    MoveL Target_890,v300,z100,PenPineappleApplePen\WObj:=krzywik;
    MoveL Target_900,v300,z100,PenPineappleApplePen\WObj:=krzywik;
    MoveL Target_910,v300,z100,PenPineappleApplePen\WObj:=krzywik;
    MoveL Target_920,v300,z100,PenPineappleApplePen\WObj:=krzywik;
    MoveL Target_930,v300,z100,PenPineappleApplePen\WObj:=krzywik;
    MoveL Target_940,v300,z100,PenPineappleApplePen\WObj:=krzywik;
    MoveL Target_950,v300,z100,PenPineappleApplePen\WObj:=krzywik;
    MoveL Target_960,v300,z100,PenPineappleApplePen\WObj:=krzywik;
    MoveL Target_970,v300,z100,PenPineappleApplePen\WObj:=krzywik;
    MoveL Target_980,v300,z100,PenPineappleApplePen\WObj:=krzywik;
    MoveL Target_990,v300,z100,PenPineappleApplePen\WObj:=krzywik;
    MoveL Target_1000,v300,z100,PenPineappleApplePen\WObj:=krzywik;
    MoveL Target_1010,v300,z100,PenPineappleApplePen\WObj:=krzywik;
    MoveL Target_1020,v300,z100,PenPineappleApplePen\WObj:=krzywik;
    MoveL Target_1030,v300,z100,PenPineappleApplePen\WObj:=krzywik;
    MoveL Target_1040,v300,z100,PenPineappleApplePen\WObj:=krzywik;
    MoveL Target_1050,v300,z100,PenPineappleApplePen\WObj:=krzywik;
    MoveL Target_1060,v300,z100,PenPineappleApplePen\WObj:=krzywik;
    MoveL Target_1070,v300,z100,PenPineappleApplePen\WObj:=krzywik;
    MoveL Target_1080,v300,z100,PenPineappleApplePen\WObj:=krzywik;
    MoveL Target_1090,v300,z100,PenPineappleApplePen\WObj:=krzywik;
    MoveL Target_1100,v300,z100,PenPineappleApplePen\WObj:=krzywik;
    MoveL Target_1110,v300,z100,PenPineappleApplePen\WObj:=krzywik;
    MoveL Target_1120,v300,z100,PenPineappleApplePen\WObj:=krzywik;
    MoveL Target_1130,v300,z100,PenPineappleApplePen\WObj:=krzywik;
    MoveL Target_1140,v300,z100,PenPineappleApplePen\WObj:=krzywik;
    MoveL Target_1150,v300,z100,PenPineappleApplePen\WObj:=krzywik;
    MoveL Target_1160,v300,z100,PenPineappleApplePen\WObj:=krzywik;
    MoveL Target_1170,v300,z100,PenPineappleApplePen\WObj:=krzywik;
    MoveL Target_1180,v300,z100,PenPineappleApplePen\WObj:=krzywik;
    MoveL Target_1190,v300,z100,PenPineappleApplePen\WObj:=krzywik;
    MoveL Target_1200,v300,z100,PenPineappleApplePen\WObj:=krzywik;
    MoveL Target_1210,v300,z100,PenPineappleApplePen\WObj:=krzywik;
    MoveL Target_1220,v300,z100,PenPineappleApplePen\WObj:=krzywik;
    MoveL Target_1230,v300,z100,PenPineappleApplePen\WObj:=krzywik;
    MoveL Target_1240,v300,z100,PenPineappleApplePen\WObj:=krzywik;
    MoveL Target_1250,v300,z100,PenPineappleApplePen\WObj:=krzywik;
    MoveL Target_1260,v300,z100,PenPineappleApplePen\WObj:=krzywik;
    MoveL Target_1270,v300,z100,PenPineappleApplePen\WObj:=krzywik;
    MoveL Target_1280,v300,z100,PenPineappleApplePen\WObj:=krzywik;
    MoveL Target_1290,v300,z100,PenPineappleApplePen\WObj:=krzywik;
    MoveL Target_1300,v300,z100,PenPineappleApplePen\WObj:=krzywik;
    MoveL Target_1310,v300,z100,PenPineappleApplePen\WObj:=krzywik;
    MoveL Target_1320,v300,z100,PenPineappleApplePen\WObj:=krzywik;
    MoveL Target_1330,v300,z100,PenPineappleApplePen\WObj:=krzywik;
    MoveL Target_1340,v300,z100,PenPineappleApplePen\WObj:=krzywik;
    MoveL Target_1350,v300,z100,PenPineappleApplePen\WObj:=krzywik;
    MoveL Target_1360,v300,z100,PenPineappleApplePen\WObj:=krzywik;
    MoveL Target_1370,v300,z100,PenPineappleApplePen\WObj:=krzywik;
    MoveL Target_1380,v300,fine,PenPineappleApplePen\WObj:=krzywik;
    MoveL Target_1390,v300,z100,PenPineappleApplePen\WObj:=krzywik;
    MoveL above_krzywik,v1000,z100,PenPineappleApplePen\WObj:=krzywik;
  ENDPROC
  PROC Path_30()
    MoveL above_lamp,v1000,z100,PenPineappleApplePen\WObj:=lampa;
    MoveL Target_1640,v300,z100,PenPineappleApplePen\WObj:=lampa;
    MoveL Target_1630,v50,fine,PenPineappleApplePen\WObj:=lampa;
    MoveL Target_1620,v50,z100,PenPineappleApplePen\WObj:=lampa;
    MoveL Target_1610,v50,z100,PenPineappleApplePen\WObj:=lampa;
    MoveL Target_1600,v50,z100,PenPineappleApplePen\WObj:=lampa;
    MoveL Target_1590,v50,z100,PenPineappleApplePen\WObj:=lampa;
    MoveL Target_1580,v50,z100,PenPineappleApplePen\WObj:=lampa;
    MoveL Target_1570,v50,z100,PenPineappleApplePen\WObj:=lampa;
    MoveL Target_1560,v50,z100,PenPineappleApplePen\WObj:=lampa;
    MoveL Target_1550,v50,z100,PenPineappleApplePen\WObj:=lampa;
    MoveL Target_1540,v50,z100,PenPineappleApplePen\WObj:=lampa;
    MoveL Target_1530,v50,z100,PenPineappleApplePen\WObj:=lampa;
    MoveL Target_1520,v50,z100,PenPineappleApplePen\WObj:=lampa;
    MoveL Target_1510,v50,z100,PenPineappleApplePen\WObj:=lampa;
    MoveL Target_1500,v50,z100,PenPineappleApplePen\WObj:=lampa;
    MoveL Target_1490,v50,z100,PenPineappleApplePen\WObj:=lampa;
    MoveL Target_1480,v50,z100,PenPineappleApplePen\WObj:=lampa;
    MoveL Target_1470,v50,z100,PenPineappleApplePen\WObj:=lampa;
    MoveL back_trace,v1000,z100,PenPineappleApplePen\WObj:=lampa;
    MoveL above_lamp,v1000,z100,PenPineappleApplePen\WObj:=lampa;
  ENDPROC
  LOCAL PROC main()
    Path_10;
  ENDPROC
ENDMODULE


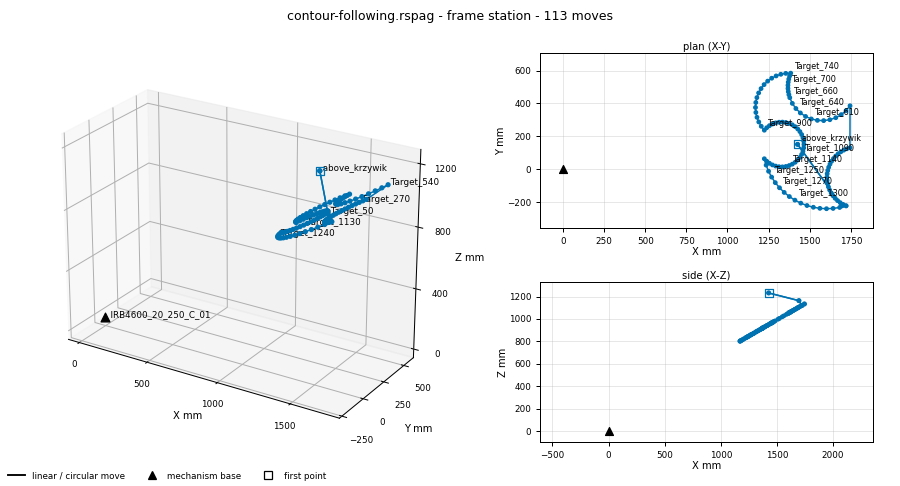
[picture p0: tool path of contour-following.rspag in frame station, 113 of 113 moves have a stored position in this frame; points joined in program order, loops and branches not executed]
--- Backups/Controller2/RAPID/TASK1/PROGMOD/RsTempModule.mod ---
MODULE RsTempModule
    LOCAL CONST robtarget above_krzywik:=[[1426.339310131,151.258623383,1181.823410703],[0.355319487,-0.049345838,0.933252419,0.018787562],[0,0,-1,1],[9E+09,9E+09,9E+09,9E+09,9E+09,9E+09]];
    LOCAL PERS tooldata PenPineappleApplePen:=[TRUE,[[56.855,0,134.138],[0.924076443,0,0.382207702,0]],[2,[2.491,0,42.7],[1,0,0,0],0,0,0]];
    LOCAL PERS wobjdata krzywik:=[FALSE,TRUE,"",[[0,0,50],[1,0,0,0]],[[0,0,0],[1,0,0,0]]];
    LOCAL CONST robtarget Target_50:=[[1696,-222.478,1113.035363495],[0.355319487,-0.049345838,0.933252419,0.018787562],[-1,-1,0,1],[9E+09,9E+09,9E+09,9E+09,9E+09,9E+09]];
    LOCAL CONST robtarget Target_60:=[[1721,-222.478,1069.734093306],[0.355319487,-0.049345838,0.933252419,0.018787562],[-1,-1,0,1],[9E+09,9E+09,9E+09,9E+09,9E+09,9E+09]];
    LOCAL CONST robtarget Target_70:=[[1702.669888124,-213.854656131,1059.15119828],[0.355319487,-0.049345838,0.933252419,0.018787562],[-1,-1,0,1],[9E+09,9E+09,9E+09,9E+09,9E+09,9E+09]];
    LOCAL CONST robtarget Target_80:=[[1685.385723439,-203.289964368,1049.172181146],[0.355319487,-0.049345838,0.933252419,0.018787562],[-1,-1,0,1],[9E+09,9E+09,9E+09,9E+09,9E+09,9E+09]];
    LOCAL CONST robtarget Target_90:=[[1669.352328762,-190.909119647,1039.915296413],[0.355319487,-0.049345838,0.933252419,0.018787562],[-1,-1,0,1],[9E+09,9E+09,9E+09,9E+09,9E+09,9E+09]];
    LOCAL CONST robtarget Target_100:=[[1654.759704885,-176.858838892,1031.49024109],[0.355319487,-0.049345838,0.933252419,0.018787562],[-1,-1,0,1],[9E+09,9E+09,9E+09,9E+09,9E+09,9E+09]];
    LOCAL CONST robtarget Target_110:=[[1641.780779016,-161.30562237,1023.996854746],[0.355319487,-0.049345838,0.933252419,0.018787562],[-1,-1,0,1],[9E+09,9E+09,9E+09,9E+09,9E+09,9E+09]];
    LOCAL CONST robtarget Target_120:=[[1630.569355527,-144.433780614,1017.523936376],[0.355319487,-0.049345838,0.933252419,0.018787562],[-1,-1,0,1],[9E+09,9E+09,9E+09,9E+09,9E+09,9E+09]];
    LOCAL CONST robtarget Target_130:=[[1621.25829333,-126.443250281,1012.148192111],[0.355319487,-0.049345838,0.933252419,0.018787562],[-1,-1,0,1],[9E+09,9E+09,9E+09,9E+09,9E+09,9E+09]];
    LOCAL CONST robtarget Target_140:=[[1613.957931457,-107.547224842,1007.933326218],[0.355319487,-0.049345838,0.933252419,0.018787562],[-1,-1,0,1],[9E+09,9E+09,9E+09,9E+09,9E+09,9E+09]];
    LOCAL CONST robtarget Target_150:=[[1608.754781501,-87.969628171,1004.92928619],[0.355319487,-0.049345838,0.933252419,0.018787562],[-1,-1,0,1],[9E+09,9E+09,9E+09,9E+09,9E+09,9E+09]];
    LOCAL CONST robtarget Target_160:=[[1605.710502435,-67.942460975,1003.171670852],[0.355319487,-0.049345838,0.933252419,0.018787562],[-1,-1,0,1],[9E+09,9E+09,9E+09,9E+09,9E+09,9E+09]];
    LOCAL CONST robtarget Target_170:=[[1604.861169929,-47.703051518,1002.681308501],[0.355319487,-0.049345838,0.933252419,0.018787562],[-1,-1,0,1],[9E+09,9E+09,9E+09,9E+09,9E+09,9E+09]];
    LOCAL CONST robtarget Target_180:=[[1606.21684884,-27.491243198,1003.464010085],[0.355319487,-0.049345838,0.933252419,0.018787562],[-1,-1,0,1],[9E+09,9E+09,9E+09,9E+09,9E+09,9E+09]];
    LOCAL CONST robtarget Target_190:=[[1609.761473944,-7.546552331,1005.510500343],[0.355319487,-0.049345838,0.933252419,0.018787562],[-1,-1,0,1],[9E+09,9E+09,9E+09,9E+09,9E+09,9E+09]];
    LOCAL CONST robtarget Target_200:=[[1615.453040316,11.89467019,1008.79652772],[0.355319487,-0.049345838,0.933252419,0.018787562],[-1,-1,0,1],[9E+09,9E+09,9E+09,9E+09,9E+09,9E+09]];
    LOCAL CONST robtarget Target_210:=[[1623.224101092,30.602039735,1013.283151751],[0.355319487,-0.049345838,0.933252419,0.018787562],[0,-1,0,1],[9E+09,9E+09,9E+09,9E+09,9E+09,9E+09]];
    LOCAL CONST robtarget Target_220:=[[1632.982566748,48.353868061,1018.917204525],[0.355319487,-0.049345838,0.933252419,0.018787562],[0,-1,0,1],[9E+09,9E+09,9E+09,9E+09,9E+09,9E+09]];
    LOCAL CONST robtarget Target_230:=[[1644.612796381,64.939790393,1025.631920734],[0.355319487,-0.049345838,0.933252419,0.018787562],[0,-1,0,1],[9E+09,9E+09,9E+09,9E+09,9E+09,9E+09]];
    LOCAL CONST robtarget Target_240:=[[1657.976968094,80.163258307,1033.34772887],[0.355319487,-0.049345838,0.933252419,0.018787562],[0,-1,0,1],[9E+09,9E+09,9E+09,9E+09,9E+09,9E+09]];
    LOCAL CONST robtarget Target_250:=[[1672.916712227,93.843868897,1041.973194167],[0.355319487,-0.049345838,0.933252419,0.018787562],[0,-1,0,1],[9E+09,9E+09,9E+09,9E+09,9E+09,9E+09]];
    LOCAL CONST robtarget Target_260:=[[1689.254988092,105.819502603,1051.406102135],[0.355319487,-0.049345838,0.933252419,0.018787562],[0,-1,0,1],[9E+09,9E+09,9E+09,9E+09,9E+09,9E+09]];
    LOCAL CONST robtarget Target_270:=[[1706.798181953,115.948244382,1061.534669833],[0.355319487,-0.049345838,0.933252419,0.018787562],[0,-1,0,1],[9E+09,9E+09,9E+09,9E+09,9E+09,9E+09]];
    LOCAL CONST robtarget Target_280:=[[1725.33840142,124.110065441,1072.238870534],[0.355319487,-0.049345838,0.933252419,0.018787562],[0,-1,0,1],[9E+09,9E+09,9E+09,9E+09,9E+09,9E+09]];
    LOCAL CONST robtarget Target_290:=[[1744.655939032,130.208245622,1083.391856074],[0.355319487,-0.049345838,0.933252419,0.018787562],[0,-1,0,1],[9E+09,9E+09,9E+09,9E+09,9E+09,9E+09]];
    LOCAL CONST robtarget Target_540:=[[1745.1875,385.5845,1083.698752942],[0.355319487,-0.049345838,0.933252419,0.018787562],[0,0,-1,1],[9E+09,9E+09,9E+09,9E+09,9E+09,9E+09]];
    LOCAL CONST robtarget Target_550:=[[1720.944864766,356.220958453,1069.702260964],[0.355319487,-0.049345838,0.933252419,0.018787562],[0,0,-1,1],[9E+09,9E+09,9E+09,9E+09,9E+09,9E+09]];
    LOCAL CONST robtarget Target_560:=[[1691.727205325,331.802700693,1052.83343742],[0.355319487,-0.049345838,0.933252419,0.018787562],[0,0,-1,1],[9E+09,9E+09,9E+09,9E+09,9E+09,9E+09]];
    LOCAL CONST robtarget Target_570:=[[1658.526094744,313.158420299,1033.664767289],[0.355319487,-0.049345838,0.933252419,0.018787562],[0,0,-1,1],[9E+09,9E+09,9E+09,9E+09,9E+09,9E+09]];
    LOCAL CONST robtarget Target_580:=[[1622.468294293,300.920856738,1012.846786492],[0.355319487,-0.049345838,0.933252419,0.018787562],[0,0,-1,1],[9E+09,9E+09,9E+09,9E+09,9E+09,9E+09]];
    LOCAL CONST robtarget Target_590:=[[1584.777514033,295.505321802,991.086004363],[0.355319487,-0.049345838,0.933252419,0.018787562],[0,0,-1,1],[9E+09,9E+09,9E+09,9E+09,9E+09,9E+09]];
    LOCAL CONST robtarget Target_600:=[[1546.732883206,297.095604975,969.120926514],[0.355319487,-0.049345838,0.933252419,0.018787562],[0,0,-1,1],[9E+09,9E+09,9E+09,9E+09,9E+09,9E+09]];
    LOCAL CONST robtarget Target_610:=[[1509.625539846,305.63773609,947.696991836],[0.355319487,-0.049345838,0.933252419,0.018787562],[0,0,-1,1],[9E+09,9E+09,9E+09,9E+09,9E+09,9E+09]];
    LOCAL CONST robtarget Target_620:=[[1474.714812829,320.841816939,927.541274195],[0.355319487,-0.049345838,0.933252419,0.018787562],[0,0,-1,1],[9E+09,9E+09,9E+09,9E+09,9E+09,9E+09]];
    LOCAL CONST robtarget Target_630:=[[1443.185483462,342.191859676,909.337807398],[0.355319487,-0.049345838,0.933252419,0.018787562],[0,0,-1,1],[9E+09,9E+09,9E+09,9E+09,9E+09,9E+09]];
    LOCAL CONST robtarget Target_640:=[[1416.10757701,368.96329814,893.704370819],[0.355319487,-0.049345838,0.933252419,0.018787562],[0,0,-1,1],[9E+09,9E+09,9E+09,9E+09,9E+09,9E+09]];
    LOCAL CONST robtarget Target_650:=[[1394.400048766,400.247577783,881.171523543],[0.355319487,-0.049345838,0.933252419,0.018787562],[0,0,-1,1],[9E+09,9E+09,9E+09,9E+09,9E+09,9E+09]];
    LOCAL CONST robtarget Target_660:=[[1378.799597041,434.982989703,872.164598541],[0.355319487,-0.049345838,0.933252419,0.018787562],[0,0,-1,1],[9E+09,9E+09,9E+09,9E+09,9E+09,9E+09]];
    LOCAL CONST robtarget Target_670:=[[1373.463613228,453.279987933,869.08386685],[0.355319487,-0.049345838,0.933252419,0.018787562],[0,0,-1,1],[9E+09,9E+09,9E+09,9E+09,9E+09,9E+09]];
    LOCAL CONST robtarget Target_680:=[[1369.835661499,471.990702344,866.989267943],[0.355319487,-0.049345838,0.933252419,0.018787562],[0,0,-1,1],[9E+09,9E+09,9E+09,9E+09,9E+09,9E+09]];
    LOCAL CONST robtarget Target_690:=[[1367.946588288,490.95604626,865.898611015],[0.355319487,-0.049345838,0.933252419,0.018787562],[0,0,-1,1],[9E+09,9E+09,9E+09,9E+09,9E+09,9E+09]];
    LOCAL CONST robtarget Target_700:=[[1367.812455319,510.014768039,865.82116931],[0.355319487,-0.049345838,0.933252419,0.018787562],[0,0,-1,1],[9E+09,9E+09,9E+09,9E+09,9E+09,9E+09]];
    LOCAL CONST robtarget Target_710:=[[1369.43440305,529.004822095,866.757601269],[0.355319487,-0.049345838,0.933252419,0.018787562],[0,0,-1,1],[9E+09,9E+09,9E+09,9E+09,9E+09,9E+09]];
    LOCAL CONST robtarget Target_720:=[[1372.798640973,547.764746686,868.699944939],[0.355319487,-0.049345838,0.933252419,0.018787562],[0,0,-1,1],[9E+09,9E+09,9E+09,9E+09,9E+09,9E+09]];
    LOCAL CONST robtarget Target_730:=[[1377.876564866,566.135036734,871.631685666],[0.355319487,-0.049345838,0.933252419,0.018787562],[0,0,-1,1],[9E+09,9E+09,9E+09,9E+09,9E+09,9E+09]];
    LOCAL CONST robtarget Target_740:=[[1384.625,583.9595,875.527896507],[0.355319487,-0.049345838,0.933252419,0.018787562],[0,0,-1,1],[9E+09,9E+09,9E+09,9E+09,9E+09,9E+09]];
    LOCAL CONST robtarget Target_750:=[[1354.328871964,582.733933377,858.03641883],[0.355319487,-0.049345838,0.933252419,0.018787562],[0,0,-1,1],[9E+09,9E+09,9E+09,9E+09,9E+09,9E+09]];
    LOCAL CONST robtarget Target_760:=[[1324.534785103,577.106342805,840.834794761],[0.355319487,-0.049345838,0.933252419,0.018787562],[0,0,-1,1],[9E+09,9E+09,9E+09,9E+09,9E+09,9E+09]];
    LOCAL CONST robtarget Target_770:=[[1295.878894374,567.196887017,824.290308534],[0.355319487,-0.049345838,0.933252419,0.018787562],[0,0,-1,1],[9E+09,9E+09,9E+09,9E+09,9E+09,9E+09]];
    LOCAL CONST robtarget Target_780:=[[1268.973052289,553.217149921,808.756213364],[0.355319487,-0.049345838,0.933252419,0.018787562],[0,0,-1,1],[9E+09,9E+09,9E+09,9E+09,9E+09,9E+09]];
    LOCAL CONST robtarget Target_790:=[[1244.391744818,535.46562293,794.564188878],[0.355319487,-0.049345838,0.933252419,0.018787562],[0,0,-1,1],[9E+09,9E+09,9E+09,9E+09,9E+09,9E+09]];
    LOCAL CONST robtarget Target_800:=[[1222.659825117,514.321331652,782.017259189],[0.355319487,-0.049345838,0.933252419,0.018787562],[0,0,-1,1],[9E+09,9E+09,9E+09,9E+09,9E+09,9E+09]];
    LOCAL CONST robtarget Target_810:=[[1204.24130702,490.235743044,771.383322808],[0.355319487,-0.049345838,0.933252419,0.018787562],[0,0,-1,1],[9E+09,9E+09,9E+09,9E+09,9E+09,9E+09]];
    LOCAL CONST robtarget Target_820:=[[1189.529457541,463.723125813,762.889432551],[0.355319487,-0.049345838,0.933252419,0.018787562],[0,0,-1,1],[9E+09,9E+09,9E+09,9E+09,9E+09,9E+09]];
    LOCAL CONST robtarget Target_830:=[[1178.83839995,435.349569901,756.716947572],[0.355319487,-0.049345838,0.933252419,0.018787562],[0,0,-1,1],[9E+09,9E+09,9E+09,9E+09,9E+09,9E+09]];
    LOCAL CONST robtarget Target_840:=[[1172.396406698,405.720899487,752.997661035],[0.355319487,-0.049345838,0.933252419,0.018787562],[0,0,-1,1],[9E+09,9E+09,9E+09,9E+09,9E+09,9E+09]];
    LOCAL CONST robtarget Target_850:=[[1170.341025414,375.469737604,751.810986097],[0.355319487,-0.049345838,0.933252419,0.018787562],[0,0,-1,1],[9E+09,9E+09,9E+09,9E+09,9E+09,9E+09]];
    LOCAL CONST robtarget Target_860:=[[1172.716142018,345.241998545,753.182260308],[0.355319487,-0.049345838,0.933252419,0.018787562],[0,0,-1,1],[9E+09,9E+09,9E+09,9E+09,9E+09,9E+09]];
    LOCAL CONST robtarget Target_870:=[[1179.471043691,315.683096486,757.082204607],[0.355319487,-0.049345838,0.933252419,0.018787562],[0,0,-1,1],[9E+09,9E+09,9E+09,9E+09,9E+09,9E+09]];
    LOCAL CONST robtarget Target_880:=[[1190.461501673,287.424164785,763.427548481],[0.355319487,-0.049345838,0.933252419,0.018787562],[0,0,-1,1],[9E+09,9E+09,9E+09,9E+09,9E+09,9E+09]];
    LOCAL CONST robtarget Target_890:=[[1205.452850798,261.068580198,772.082807934],[0.355319487,-0.049345838,0.933252419,0.018787562],[0,0,-1,1],[9E+09,9E+09,9E+09,9E+09,9E+09,9E+09]];
    LOCAL CONST robtarget Target_900:=[[1224.125,237.179079749,782.863178302],[0.355319487,-0.049345838,0.933252419,0.018787562],[0,0,-1,1],[9E+09,9E+09,9E+09,9E+09,9E+09,9E+09]];
    LOCAL CONST robtarget Target_910:=[[1238.592084328,252.176181987,791.215753333],[0.355319487,-0.049345838,0.933252419,0.018787562],[0,0,-1,1],[9E+09,9E+09,9E+09,9E+09,9E+09,9E+09]];
    LOCAL CONST robtarget Target_920:=[[1255.177965809,264.790385883,800.791616471],[0.355319487,-0.049345838,0.933252419,0.018787562],[0,0,-1,1],[9E+09,9E+09,9E+09,9E+09,9E+09,9E+09]];
    LOCAL CONST robtarget Target_930:=[[1273.49426739,274.726315678,811.366538119],[0.355319487,-0.049345838,0.933252419,0.018787562],[0,0,-1,1],[9E+09,9E+09,9E+09,9E+09,9E+09,9E+09]];
    LOCAL CONST robtarget Target_940:=[[1293.112092282,281.751310408,822.692894602],[0.355319487,-0.049345838,0.933252419,0.018787562],[0,0,-1,1],[9E+09,9E+09,9E+09,9E+09,9E+09,9E+09]];
    LOCAL CONST robtarget Target_950:=[[1313.572067069,285.700871927,834.505466553],[0.355319487,-0.049345838,0.933252419,0.018787562],[0,0,-1,1],[9E+09,9E+09,9E+09,9E+09,9E+09,9E+09]];
    LOCAL CONST robtarget Target_960:=[[1334.395098447,286.482516812,846.527649324],[0.355319487,-0.049345838,0.933252419,0.018787562],[0,0,-1,1],[9E+09,9E+09,9E+09,9E+09,9E+09,9E+09]];
    LOCAL CONST robtarget Target_970:=[[1355.093591733,284.07794197,858.477929994],[0.355319487,-0.049345838,0.933252419,0.018787562],[0,0,-1,1],[9E+09,9E+09,9E+09,9E+09,9E+09,9E+09]];
    LOCAL CONST robtarget Target_980:=[[1375.182868444,278.543453224,870.076479312],[0.355319487,-0.049345838,0.933252419,0.018787562],[0,0,-1,1],[9E+09,9E+09,9E+09,9E+09,9E+09,9E+09]];
    LOCAL CONST robtarget Target_990:=[[1394.192515589,270.008646848,881.051704208],[0.355319487,-0.049345838,0.933252419,0.018787562],[0,0,-1,1],[9E+09,9E+09,9E+09,9E+09,9E+09,9E+09]];
    LOCAL CONST robtarget Target_1000:=[[1411.677400916,258.673374924,891.146607458],[0.355319487,-0.049345838,0.933252419,0.018787562],[0,0,-1,1],[9E+09,9E+09,9E+09,9E+09,9E+09,9E+09]];
    LOCAL CONST robtarget Target_1010:=[[1427.228096184,244.803065585,900.124805557],[0.355319487,-0.049345838,0.933252419,0.018787562],[0,0,-1,1],[9E+09,9E+09,9E+09,9E+09,9E+09,9E+09]];
    LOCAL CONST robtarget Target_1020:=[[1440.480464386,228.722507712,907.776063906],[0.355319487,-0.049345838,0.933252419,0.018787562],[0,0,-1,1],[9E+09,9E+09,9E+09,9E+09,9E+09,9E+09]];
    LOCAL CONST robtarget Target_1030:=[[1451.124186427,210.80824564,913.921219691],[0.355319487,-0.049345838,0.933252419,0.018787562],[0,0,-1,1],[9E+09,9E+09,9E+09,9E+09,9E+09,9E+09]];
    LOCAL CONST robtarget Target_1040:=[[1458.910027592,191.479761948,918.416377184],[0.355319487,-0.049345838,0.933252419,0.018787562],[0,0,-1,1],[9E+09,9E+09,9E+09,9E+09,9E+09,9E+09]];
    LOCAL CONST robtarget Target_1050:=[[1463.655673662,171.189654806,921.15627722],[0.355319487,-0.049345838,0.933252419,0.018787562],[0,0,-1,1],[9E+09,9E+09,9E+09,9E+09,9E+09,9E+09]];
    LOCAL CONST robtarget Target_1060:=[[1465.25,150.413039874,922.076761961],[0.355319487,-0.049345838,0.933252419,0.018787562],[0,-1,0,1],[9E+09,9E+09,9E+09,9E+09,9E+09,9E+09]];
    LOCAL CONST robtarget Target_1070:=[[1463.655673662,129.636424943,921.15627722],[0.355319487,-0.049345838,0.933252419,0.018787562],[0,-1,0,1],[9E+09,9E+09,9E+09,9E+09,9E+09,9E+09]];
    LOCAL CONST robtarget Target_1080:=[[1458.910027592,109.346317801,918.416377184],[0.355319487,-0.049345838,0.933252419,0.018787562],[0,-1,0,1],[9E+09,9E+09,9E+09,9E+09,9E+09,9E+09]];
    LOCAL CONST robtarget Target_1090:=[[1451.124186427,90.017834109,913.921219691],[0.355319487,-0.049345838,0.933252419,0.018787562],[0,-1,0,1],[9E+09,9E+09,9E+09,9E+09,9E+09,9E+09]];
    LOCAL CONST robtarget Target_1100:=[[1440.480464386,72.103572037,907.776063906],[0.355319487,-0.049345838,0.933252419,0.018787562],[0,-1,0,1],[9E+09,9E+09,9E+09,9E+09,9E+09,9E+09]];
    LOCAL CONST robtarget Target_1110:=[[1427.228096184,56.023014164,900.124805557],[0.355319487,-0.049345838,0.933252419,0.018787562],[0,-1,0,1],[9E+09,9E+09,9E+09,9E+09,9E+09,9E+09]];
    LOCAL CONST robtarget Target_1120:=[[1411.677400916,42.152704825,891.146607458],[0.355319487,-0.049345838,0.933252419,0.018787562],[0,-1,0,1],[9E+09,9E+09,9E+09,9E+09,9E+09,9E+09]];
    LOCAL CONST robtarget Target_1130:=[[1394.192515589,30.817432901,881.051704208],[0.355319487,-0.049345838,0.933252419,0.018787562],[0,-1,0,1],[9E+09,9E+09,9E+09,9E+09,9E+09,9E+09]];
    LOCAL CONST robtarget Target_1140:=[[1375.182868444,22.282626525,870.076479312],[0.355319487,-0.049345838,0.933252419,0.018787562],[-1,-1,0,1],[9E+09,9E+09,9E+09,9E+09,9E+09,9E+09]];
    LOCAL CONST robtarget Target_1150:=[[1355.093591733,16.748137779,858.477929994],[0.355319487,-0.049345838,0.933252419,0.018787562],[-1,-1,0,1],[9E+09,9E+09,9E+09,9E+09,9E+09,9E+09]];
    LOCAL CONST robtarget Target_1160:=[[1334.395098447,14.343562937,846.527649324],[0.355319487,-0.049345838,0.933252419,0.018787562],[-1,-1,0,1],[9E+09,9E+09,9E+09,9E+09,9E+09,9E+09]];
    LOCAL CONST robtarget Target_1170:=[[1313.572067069,15.125207822,834.505466553],[0.355319487,-0.049345838,0.933252419,0.018787562],[-1,-1,0,1],[9E+09,9E+09,9E+09,9E+09,9E+09,9E+09]];
    LOCAL CONST robtarget Target_1180:=[[1293.112092282,19.074769341,822.692894602],[0.355319487,-0.049345838,0.933252419,0.018787562],[-1,-1,0,1],[9E+09,9E+09,9E+09,9E+09,9E+09,9E+09]];
    LOCAL CONST robtarget Target_1190:=[[1273.49426739,26.099764071,811.366538119],[0.355319487,-0.049345838,0.933252419,0.018787562],[0,-1,0,1],[9E+09,9E+09,9E+09,9E+09,9E+09,9E+09]];
    LOCAL CONST robtarget Target_1200:=[[1255.177965809,36.035693866,800.791616471],[0.355319487,-0.049345838,0.933252419,0.018787562],[0,-1,0,1],[9E+09,9E+09,9E+09,9E+09,9E+09,9E+09]];
    LOCAL CONST robtarget Target_1210:=[[1238.592084328,48.649897762,791.215753333],[0.355319487,-0.049345838,0.933252419,0.018787562],[0,-1,0,1],[9E+09,9E+09,9E+09,9E+09,9E+09,9E+09]];
    LOCAL CONST robtarget Target_1220:=[[1224.125,63.647,782.863178302],[0.355319487,-0.049345838,0.933252419,0.018787562],[0,-1,0,1],[9E+09,9E+09,9E+09,9E+09,9E+09,9E+09]];
    LOCAL CONST robtarget Target_1230:=[[1235.068705531,24.942095166,789.181529636],[0.355319487,-0.049345838,0.933252419,0.018787562],[0,-1,0,1],[9E+09,9E+09,9E+09,9E+09,9E+09,9E+09]];
    LOCAL CONST robtarget Target_1240:=[[1249.93531583,-12.431936557,797.764771094],[0.355319487,-0.049345838,0.933252419,0.018787562],[-1,-1,0,1],[9E+09,9E+09,9E+09,9E+09,9E+09,9E+09]];
    LOCAL CONST robtarget Target_1250:=[[1268.567140429,-48.078667979,808.521860042],[0.355319487,-0.049345838,0.933252419,0.018787562],[-1,-1,0,1],[9E+09,9E+09,9E+09,9E+09,9E+09,9E+09]];
    LOCAL CONST robtarget Target_1260:=[[1290.76655115,-81.619993425,821.338695798],[0.355319487,-0.049345838,0.933252419,0.018787562],[-1,-1,0,1],[9E+09,9E+09,9E+09,9E+09,9E+09,9E+09]];
    LOCAL CONST robtarget Target_1270:=[[1316.298078347,-112.700139306,836.079329898],[0.355319487,-0.049345838,0.933252419,0.018787562],[-1,-1,0,1],[9E+09,9E+09,9E+09,9E+09,9E+09,9E+09]];
    LOCAL CONST robtarget Target_1280:=[[1344.890908541,-140.989437821,852.587408107],[0.355319487,-0.049345838,0.933252419,0.018787562],[-1,-1,0,1],[9E+09,9E+09,9E+09,9E+09,9E+09,9E+09]];
    LOCAL CONST robtarget Target_1290:=[[1376.241756944,-166.187823749,870.687828872],[0.355319487,-0.049345838,0.933252419,0.018787562],[-1,-1,0,1],[9E+09,9E+09,9E+09,9E+09,9E+09,9E+09]];
    LOCAL CONST robtarget Target_1300:=[[1410.018084407,-188.028017249,890.188600625],[0.355319487,-0.049345838,0.933252419,0.018787562],[-1,-1,0,1],[9E+09,9E+09,9E+09,9E+09,9E+09,9E+09]];
    LOCAL CONST robtarget Target_1310:=[[1445.86162467,-206.2783589,910.882878245],[0.355319487,-0.049345838,0.933252419,0.018787562],[-1,-1,0,1],[9E+09,9E+09,9E+09,9E+09,9E+09,9E+09]];
    LOCAL CONST robtarget Target_1320:=[[1483.392184502,-220.745266921,932.551157066],[0.355319487,-0.049345838,0.933252419,0.018787562],[-1,-1,0,1],[9E+09,9E+09,9E+09,9E+09,9E+09,9E+09]];
    LOCAL CONST robtarget Target_1330:=[[1522.211676416,-231.275290496,954.963601173],[0.355319487,-0.049345838,0.933252419,0.018787562],[-1,-1,0,1],[9E+09,9E+09,9E+09,9E+09,9E+09,9E+09]];
    LOCAL CONST robtarget Target_1340:=[[1561.908341196,-237.756737429,977.88248127],[0.355319487,-0.049345838,0.933252419,0.018787562],[-1,-1,0,1],[9E+09,9E+09,9E+09,9E+09,9E+09,9E+09]];
    LOCAL CONST robtarget Target_1350:=[[1602.061115432,-240.120858867,1001.064696283],[0.355319487,-0.049345838,0.933252419,0.018787562],[-1,-1,0,1],[9E+09,9E+09,9E+09,9E+09,9E+09,9E+09]];
    LOCAL CONST robtarget Target_1360:=[[1642.24409775,-238.342578523,1024.264351942],[0.355319487,-0.049345838,0.933252419,0.018787562],[-1,-1,0,1],[9E+09,9E+09,9E+09,9E+09,9E+09,9E+09]];
    LOCAL CONST robtarget Target_1370:=[[1682.031066361,-232.440758656,1047.235368979],[0.355319487,-0.049345838,0.933252419,0.018787562],[-1,-1,0,1],[9E+09,9E+09,9E+09,9E+09,9E+09,9E+09]];
    LOCAL CONST robtarget Target_1380:=[[1721,-222.478,1069.734093306],[0.355319487,-0.049345838,0.933252419,0.018787562],[-1,-1,0,1],[9E+09,9E+09,9E+09,9E+09,9E+09,9E+09]];
    LOCAL CONST robtarget Target_1390:=[[1696,-222.478,1113.035363495],[0.355319487,-0.049345838,0.933252419,0.018787562],[-1,-1,0,1],[9E+09,9E+09,9E+09,9E+09,9E+09,9E+09]];
PROC RsTempPath()
        MoveL above_krzywik,v1000,z100,PenPineappleApplePen\WObj:=krzywik;
        MoveL Target_50,v1000,z100,PenPineappleApplePen\WObj:=krzywik;
        MoveL Target_60,v300,fine,PenPineappleApplePen\WObj:=krzywik;
        MoveL Target_70,v300,z100,PenPineappleApplePen\WObj:=krzywik;
        MoveL Target_80,v300,z100,PenPineappleApplePen\WObj:=krzywik;
        MoveL Target_90,v300,z100,PenPineappleApplePen\WObj:=krzywik;
        MoveL Target_100,v300,z100,PenPineappleApplePen\WObj:=krzywik;
        MoveL Target_110,v300,z100,PenPineappleApplePen\WObj:=krzywik;
        MoveL Target_120,v300,z100,PenPineappleApplePen\WObj:=krzywik;
        MoveL Target_130,v300,z100,PenPineappleApplePen\WObj:=krzywik;
        MoveL Target_140,v300,z100,PenPineappleApplePen\WObj:=krzywik;
        MoveL Target_150,v300,z100,PenPineappleApplePen\WObj:=krzywik;
        MoveL Target_160,v300,z100,PenPineappleApplePen\WObj:=krzywik;
        MoveL Target_170,v300,z100,PenPineappleApplePen\WObj:=krzywik;
        MoveL Target_180,v300,z100,PenPineappleApplePen\WObj:=krzywik;
        MoveL Target_190,v300,z100,PenPineappleApplePen\WObj:=krzywik;
        MoveL Target_200,v300,z100,PenPineappleApplePen\WObj:=krzywik;
        MoveL Target_210,v300,z100,PenPineappleApplePen\WObj:=krzywik;
        MoveL Target_220,v300,z100,PenPineappleApplePen\WObj:=krzywik;
        MoveL Target_230,v300,z100,PenPineappleApplePen\WObj:=krzywik;
        MoveL Target_240,v300,z100,PenPineappleApplePen\WObj:=krzywik;
        MoveL Target_250,v300,z100,PenPineappleApplePen\WObj:=krzywik;
        MoveL Target_260,v300,z100,PenPineappleApplePen\WObj:=krzywik;
        MoveL Target_270,v300,z100,PenPineappleApplePen\WObj:=krzywik;
        MoveL Target_280,v300,z100,PenPineappleApplePen\WObj:=krzywik;
        MoveL Target_290,v300,z100,PenPineappleApplePen\WObj:=krzywik;
        MoveL Target_540,v300,z100,PenPineappleApplePen\WObj:=krzywik;
        MoveL Target_550,v300,z100,PenPineappleApplePen\WObj:=krzywik;
        MoveL Target_560,v300,z100,PenPineappleApplePen\WObj:=krzywik;
        MoveL Target_570,v300,z100,PenPineappleApplePen\WObj:=krzywik;
        MoveL Target_580,v300,z100,PenPineappleApplePen\WObj:=krzywik;
        MoveL Target_590,v300,z100,PenPineappleApplePen\WObj:=krzywik;
        MoveL Target_600,v300,z100,PenPineappleApplePen\WObj:=krzywik;
        MoveL Target_610,v300,z100,PenPineappleApplePen\WObj:=krzywik;
        MoveL Target_620,v300,z100,PenPineappleApplePen\WObj:=krzywik;
        MoveL Target_630,v300,z100,PenPineappleApplePen\WObj:=krzywik;
        MoveL Target_640,v300,z100,PenPineappleApplePen\WObj:=krzywik;
        MoveL Target_650,v300,z100,PenPineappleApplePen\WObj:=krzywik;
        MoveL Target_660,v300,z100,PenPineappleApplePen\WObj:=krzywik;
        MoveL Target_670,v300,z100,PenPineappleApplePen\WObj:=krzywik;
        MoveL Target_680,v300,z100,PenPineappleApplePen\WObj:=krzywik;
        MoveL Target_690,v300,z100,PenPineappleApplePen\WObj:=krzywik;
        MoveL Target_700,v300,z100,PenPineappleApplePen\WObj:=krzywik;
        MoveL Target_710,v300,z100,PenPineappleApplePen\WObj:=krzywik;
        MoveL Target_720,v300,z100,PenPineappleApplePen\WObj:=krzywik;
        MoveL Target_730,v300,z100,PenPineappleApplePen\WObj:=krzywik;
        MoveL Target_740,v300,z100,PenPineappleApplePen\WObj:=krzywik;
        MoveL Target_750,v300,z100,PenPineappleApplePen\WObj:=krzywik;
        MoveL Target_760,v300,z100,PenPineappleApplePen\WObj:=krzywik;
        MoveL Target_770,v300,z100,PenPineappleApplePen\WObj:=krzywik;
        MoveL Target_780,v300,z100,PenPineappleApplePen\WObj:=krzywik;
        MoveL Target_790,v300,z100,PenPineappleApplePen\WObj:=krzywik;
        MoveL Target_800,v300,z100,PenPineappleApplePen\WObj:=krzywik;
        MoveL Target_810,v300,z100,PenPineappleApplePen\WObj:=krzywik;
        MoveL Target_820,v300,z100,PenPineappleApplePen\WObj:=krzywik;
        MoveL Target_830,v300,z100,PenPineappleApplePen\WObj:=krzywik;
        MoveL Target_840,v300,z100,PenPineappleApplePen\WObj:=krzywik;
        MoveL Target_850,v300,z100,PenPineappleApplePen\WObj:=krzywik;
        MoveL Target_860,v300,z100,PenPineappleApplePen\WObj:=krzywik;
        MoveL Target_870,v300,z100,PenPineappleApplePen\WObj:=krzywik;
        MoveL Target_880,v300,z100,PenPineappleApplePen\WObj:=krzywik;
        MoveL Target_890,v300,z100,PenPineappleApplePen\WObj:=krzywik;
        MoveL Target_900,v300,z100,PenPineappleApplePen\WObj:=krzywik;
        MoveL Target_910,v300,z100,PenPineappleApplePen\WObj:=krzywik;
        MoveL Target_920,v300,z100,PenPineappleApplePen\WObj:=krzywik;
        MoveL Target_930,v300,z100,PenPineappleApplePen\WObj:=krzywik;
        MoveL Target_940,v300,z100,PenPineappleApplePen\WObj:=krzywik;
        MoveL Target_950,v300,z100,PenPineappleApplePen\WObj:=krzywik;
        MoveL Target_960,v300,z100,PenPineappleApplePen\WObj:=krzywik;
        MoveL Target_970,v300,z100,PenPineappleApplePen\WObj:=krzywik;
        MoveL Target_980,v300,z100,PenPineappleApplePen\WObj:=krzywik;
        MoveL Target_990,v300,z100,PenPineappleApplePen\WObj:=krzywik;
        MoveL Target_1000,v300,z100,PenPineappleApplePen\WObj:=krzywik;
        MoveL Target_1010,v300,z100,PenPineappleApplePen\WObj:=krzywik;
        MoveL Target_1020,v300,z100,PenPineappleApplePen\WObj:=krzywik;
        MoveL Target_1030,v300,z100,PenPineappleApplePen\WObj:=krzywik;
        MoveL Target_1040,v300,z100,PenPineappleApplePen\WObj:=krzywik;
        MoveL Target_1050,v300,z100,PenPineappleApplePen\WObj:=krzywik;
        MoveL Target_1060,v300,z100,PenPineappleApplePen\WObj:=krzywik;
        MoveL Target_1070,v300,z100,PenPineappleApplePen\WObj:=krzywik;
        MoveL Target_1080,v300,z100,PenPineappleApplePen\WObj:=krzywik;
        MoveL Target_1090,v300,z100,PenPineappleApplePen\WObj:=krzywik;
        MoveL Target_1100,v300,z100,PenPineappleApplePen\WObj:=krzywik;
        MoveL Target_1110,v300,z100,PenPineappleApplePen\WObj:=krzywik;
        MoveL Target_1120,v300,z100,PenPineappleApplePen\WObj:=krzywik;
        MoveL Target_1130,v300,z100,PenPineappleApplePen\WObj:=krzywik;
        MoveL Target_1140,v300,z100,PenPineappleApplePen\WObj:=krzywik;
        MoveL Target_1150,v300,z100,PenPineappleApplePen\WObj:=krzywik;
        MoveL Target_1160,v300,z100,PenPineappleApplePen\WObj:=krzywik;
        MoveL Target_1170,v300,z100,PenPineappleApplePen\WObj:=krzywik;
        MoveL Target_1180,v300,z100,PenPineappleApplePen\WObj:=krzywik;
        MoveL Target_1190,v300,z100,PenPineappleApplePen\WObj:=krzywik;
        MoveL Target_1200,v300,z100,PenPineappleApplePen\WObj:=krzywik;
        MoveL Target_1210,v300,z100,PenPineappleApplePen\WObj:=krzywik;
        MoveL Target_1220,v300,z100,PenPineappleApplePen\WObj:=krzywik;
        MoveL Target_1230,v300,z100,PenPineappleApplePen\WObj:=krzywik;
        MoveL Target_1240,v300,z100,PenPineappleApplePen\WObj:=krzywik;
        MoveL Target_1250,v300,z100,PenPineappleApplePen\WObj:=krzywik;
        MoveL Target_1260,v300,z100,PenPineappleApplePen\WObj:=krzywik;
        MoveL Target_1270,v300,z100,PenPineappleApplePen\WObj:=krzywik;
        MoveL Target_1280,v300,z100,PenPineappleApplePen\WObj:=krzywik;
        MoveL Target_1290,v300,z100,PenPineappleApplePen\WObj:=krzywik;
        MoveL Target_1300,v300,z100,PenPineappleApplePen\WObj:=krzywik;
        MoveL Target_1310,v300,z100,PenPineappleApplePen\WObj:=krzywik;
        MoveL Target_1320,v300,z100,PenPineappleApplePen\WObj:=krzywik;
        MoveL Target_1330,v300,z100,PenPineappleApplePen\WObj:=krzywik;
        MoveL Target_1340,v300,z100,PenPineappleApplePen\WObj:=krzywik;
        MoveL Target_1350,v300,z100,PenPineappleApplePen\WObj:=krzywik;
        MoveL Target_1360,v300,z100,PenPineappleApplePen\WObj:=krzywik;
        MoveL Target_1370,v300,z100,PenPineappleApplePen\WObj:=krzywik;
        MoveL Target_1380,v300,fine,PenPineappleApplePen\WObj:=krzywik;
        MoveL Target_1390,v300,z100,PenPineappleApplePen\WObj:=krzywik;
        MoveL above_krzywik,v1000,z100,PenPineappleApplePen\WObj:=krzywik;
        SetSysData wobj0;
        SetSysData tool0;
ENDPROC

ENDMODULE
